ABB RobotStudio station: IRC5fisico_20230607-090725.rsstn

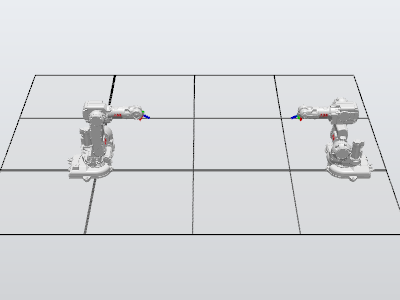
Station IRC5fisico (saved by RobotStudio 22.3.10190.2)
Layout (positions relative to the parent item):
  - IRB140_6_81_C_03 [mechanism, from Robots\IRB140_6_81_C_G_03.rslib] at (0, 0, 0) mm; joint values [0, 0, 0, 0, 0.5236, 0] (rad or m)
  - IRB140_6_81_C_03_4 [mechanism, from Robots\IRB140_6_81_C_G_03.rslib] at (2539.56, 0, 0) mm, rotated rx 0 ry 0 rz -179.36 deg; joint values [0, 0, 0, 0, 0.5236, 0] (rad or m)
